# B&R Automation Studio project Lab3
Automation Studio 4.5.2.102

## Configuration SampleText

### Task classes (Cpu.sw)
```
Cyclic#1 (cycle 2000 us, tolerance 0 us):
  ncsdcctrl <- ncsdcctrl.prg
Cyclic#4:
  Program <- Program.prg
NcDataObjects: acp10etxen <- acp10etxen.dob, Axis_Xa <- Axis_Xobj.Axis_Xa.dob, Axis_Xi <- Axis_Xobj.Axis_Xi.dob
Libraries: Acp10sdc, sys_lib, Runtime, asstring, Acp10man, Acp10par, NcGlobal, Acp10_MC, brsystem, AsBrStr, Acp10sim, AsIOTime, Library
```

### Hardware
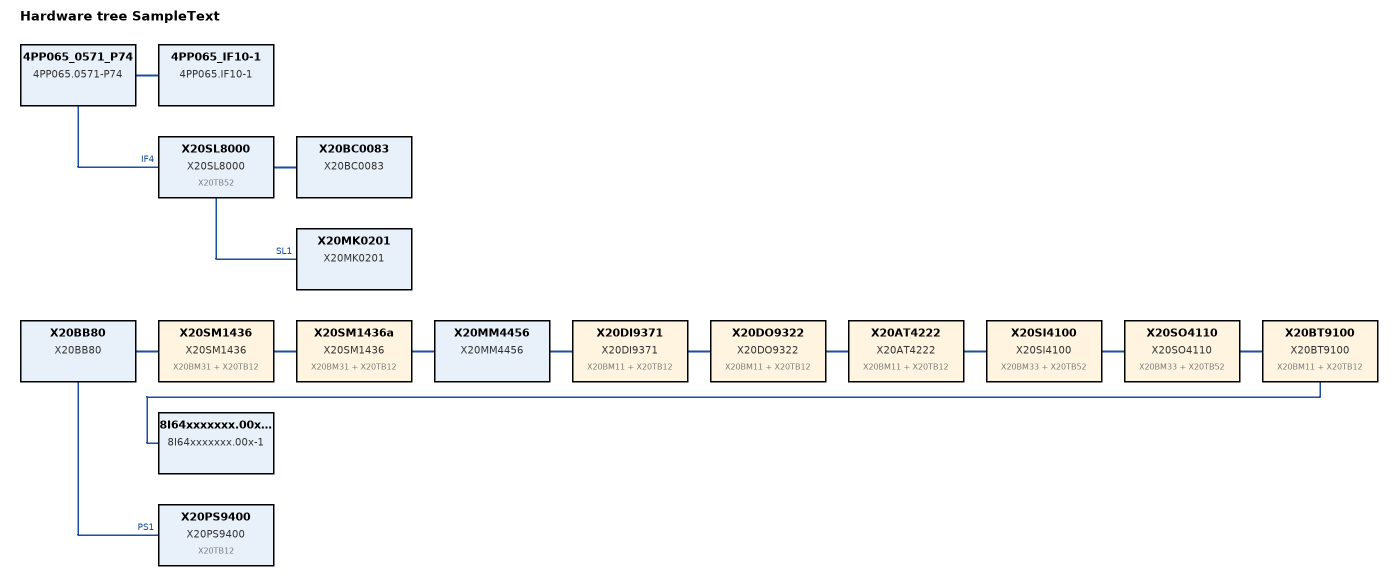
```
4PP065_0571_P74 : 4PP065.0571-P74 v1.1.2.0
  Connector IF4:
    EplInterfaceRedundant = 0
    EplEthInterfaceRedundant = 0
  Connector IF5:
    ActivateDevice = 1
    Mode = Manual
    InternetAddress = 10.1.1.13
    SubnetMask = 255.255.255.0
  ConfigurationID = DriveControl_SampleText
  Simulation = 1
  TimerDeviceType = EPLX2X
  TimerDevice = 4PP065_0571_P74.IF4
  TaskClassIdleTime = 2000
  Cyclic1Duration = 2000
  Cyclic1Tolerance = 0
  Cyclic1Output = 1
4PP065_IF10-1 : 4PP065.IF10-1 v1.0.3.0  [SS -> 4PP065_0571_P74.SS1]
8I64xxxxxxx.00x-1 : 8I64xxxxxxx.00x-1 v1.3.9.1  [X2X1 -> X20BT9100.X2X1 [Cable Type=X2XCable, Length=10, Version=1.0.0.2]]
X20AT4222 : X20AT4222 v1.2.3.0  [SS1 -> X20TB12e.SS; SL -> X20BM11c.SL1]
X20BB80 : X20BB80 v1.0.2.0
X20BC0083 : X20BC0083 v2.7.0.0  [PLK1 -> X20SL8000.PLK2 [Cable Type=PowerlinkCable, Length=10, Version=1.0.0.2]; SL -> X20BB80.SL1]
X20BM11 : X20BM11 v1.0.0.1  [X2X1 -> X20BM33a.X2X2]
X20BM11a : X20BM11 v1.0.0.1  [X2X1 -> X20MM4456.X2X2]
X20BM11b : X20BM11 v1.0.0.1  [X2X1 -> X20BM11a.X2X2]
X20BM11c : X20BM11 v1.0.0.1  [X2X1 -> X20BM11b.X2X2]
X20BM31 : X20BM31 v1.0.0.1  [X2X1 -> X20BB80.IF1]
X20BM31a : X20BM31 v1.0.0.1  [X2X1 -> X20BM31.X2X2]
X20BM33 : X20BM33 v1.0.0.4  [X2X1 -> X20BM11c.X2X2]
X20BM33a : X20BM33 v1.0.0.4  [X2X1 -> X20BM33.X2X2]
X20BT9100 : X20BT9100 v1.0.3.0  [SS1 -> X20TB12f.SS; SL -> X20BM11.SL1]
X20DI9371 : X20DI9371 v1.0.2.0  [SS1 -> X20TB12c.SS; SL -> X20BM11a.SL1]
X20DO9322 : X20DO9322 v1.0.3.0  [SS1 -> X20TB12d.SS; SL -> X20BM11b.SL1]
X20MK0201 : X20MK0201 v1.0.0.0  [SL -> X20SL8000.SL1]
X20MM4456 : X20MM4456 v1.1.5.0  [X2X1 -> X20BM31a.X2X2]
X20PS9400 : X20PS9400 v1.0.2.4  [SS1 -> X20TB12.SS; PS -> X20BB80.PS1]
X20SI4100 : X20SI4100 v1.10.1.1  [SS1 -> X20TB52.SS; SL -> X20BM33.SL1]
X20SL8000 : X20SL8000 v1.6.5.1  [PLK1 -> 4PP065_0571_P74.IF4 [Cable Type=PowerlinkCable, Length=10, Version=1.0.0.2]; PLK2 -> X20BC0083.PLK1 [Cable Type=PowerlinkCable, Length=10, Version=1.0.0.2]; SS1 -> X20TB52b.SS]
  SafeProject = SafeLOGIC-1
X20SM1436 : X20SM1436 v2.2.0.0  [SS1 -> X20TB12a.SS; SL -> X20BM31.SL1]
X20SM1436a : X20SM1436 v2.2.0.0  [SS1 -> X20TB12b.SS; SL -> X20BM31a.SL1]
X20SO4110 : X20SO4110 v1.10.1.1  [SS1 -> X20TB52a.SS; SL -> X20BM33a.SL1]
  SafeModuleID = 3
X20TB12 : X20TB12 v1.0.0.0
X20TB12a : X20TB12 v1.0.0.0
X20TB12b : X20TB12 v1.0.0.0
X20TB12c : X20TB12 v1.0.0.0
X20TB12d : X20TB12 v1.0.0.0
X20TB12e : X20TB12 v1.0.0.0
X20TB12f : X20TB12 v1.0.0.0
X20TB52 : X20TB52 v1.0.0.1
X20TB52a : X20TB52 v1.0.0.1
X20TB52b : X20TB52 v1.0.0.1
```

### IoMap.iom - 4PP065_0571_P74/IoMap.iom
```iecst
VAR_CONFIG
	Cyclic#1.Axis_X_DrvIf.iLifeCnt AT %IB."8I64xxxxxxx.00x-1".SDC_LifeCnt;
	Cyclic#1.Axis_X_DrvIf.iDrvOK AT %IX."8I64xxxxxxx.00x-1".ETAD_Input_Bool_02;
	Cyclic#1.Axis_X_DrvIf.oSetTime AT %QW."8I64xxxxxxx.00x-1".SDC_SetTime;
	Cyclic#1.Axis_X_DrvIf.oSetPos AT %QW."8I64xxxxxxx.00x-1".LFRD_Output;
	Cyclic#1.Axis_X_DiDoIf.iLifeCntDriveReady AT %IB."8I64xxxxxxx.00x-1".SDC_LifeCnt;
	Cyclic#1.Axis_X_DiDoIf.iLifeCntDriveEnable AT %IB."8I64xxxxxxx.00x-1".SDC_LifeCnt;
	Cyclic#1.Axis_X_DiDoIf.oDriveEnable AT %QX."8I64xxxxxxx.00x-1".CMDD_Output_Bool_00;
	Cyclic#1.Axis_X_ModuleOk AT %QX."8I64xxxxxxx.00x-1".CMDD_Output_Bool_01;
	Cyclic#1.Axis_X_ModuleOk AT %QX."8I64xxxxxxx.00x-1".CMDD_Output_Bool_02;
	Cyclic#1.Axis_X_ModuleOk AT %IX."8I64xxxxxxx.00x-1".ModuleOk;
	Cyclic#1.Axis_X_DiDoIf.oDriveEnable AT %QX."8I64xxxxxxx.00x-1".CMDD_Output_Bool_03;
	Cyclic#1.Axis_X_DiDoIf.iDriveReady AT %IX."8I64xxxxxxx.00x-1".ETAD_Input_Bool_02;
	::Program:coil_powered AT %IX."X20DI9371".DigitalInput01;
	::Program:axis_X.pwm_value AT %QW."X20MM4456".PulseWidthCurrentPWM01;
	::Program:axis_X.reset_error  AT %QX."X20MM4456".ClearError01;
	::Program:axis_X.endswitch_a_reached  AT %IX."X20MM4456".StatusInput03;
	::Program:axis_X.endswitch_b_reached AT %IX."X20MM4456".StatusInput04;
	::Program:axis_X.counter AT %IW."X20MM4456".Counter01;
	::Program:pwm_period  AT %QW."X20MM4456".PeriodDurationPWM;
	::Program:axis_X.reset_counter AT %QX."X20MM4456".ResetCounter01;
	::Program:coil_pwm_value  AT %QW."X20MM4456".PulseWidthCurrentPWM04;
END_VAR
```

### Acp10map.ncm - 4PP065_0571_P74/Motion/Acp10map.ncm
```
NcMapping (NcSwId=Acp10, DisabledNodesAreHidden=False)
  NcObject Axis_X (ModuleId=8I64xxxxxxx.00x-1, ModuleAddress=SDC_IF1.ST2, Type=ncAXIS, Channel=1, AcoposSimulation=Off, InitParameter=Axis_Xi, AcoposParameter=Axis_Xa, Disabled=FALSE, ModuleDisabled=FALSE)
```

## Logical view

### Axis_Xi.ax
```
InitParameter (Version=5.02.1, NcSwId=Acp10)
  ACP10AXIS_typ:
    dig_in:
      level:
        reference = ncACTIV_HI
        pos_hw_end = ncACTIV_HI
        neg_hw_end = ncACTIV_HI
        trigger1 = ncACTIV_HI
        trigger2 = ncACTIV_LO + ncQUICKSTOP
    encoder_if:
      parameter:
        count_dir = ncSTANDARD
        scaling:
          load:
            units = 3000
            rev_motor = 1
    limit:
      parameter:
        v_pos = 10000
        v_neg = 10000
        a1_pos = 10000.0
        a2_pos = 10000.0
        a1_neg = 10000.0
        a2_neg = 10000.0
        t_jolt = 0
        t_in_pos = 0
        pos_sw_end = 2000000000
        neg_sw_end = -2000000000
        ds_warning = 500
        ds_stop = 50000.0
        a_stop = 1.0e30
        dv_stop = 0
        dv_stop_mode = ncOFF
    controller:
      mode = ncPOSITION
      position:
        kv = 10.0
        tn = 0
        t_predict = 0.01
        t_total = 0.01
        p_max = 1.0e30
        i_max = 0
      speed:
        kv = 2.0
        tn = 0
        t_filter = 0.0
        isq_filter1:
          type = ncOFF
          a0 = 0.0
          a1 = 0.0
          b0 = 0.0
          b1 = 0.0
          b2 = 0.0
          c0_par_id = 0
          c1_par_id = 0
        isq_filter2:
          type = ncOFF
          a0 = 0.0
          a1 = 0.0
          b0 = 0.0
          b1 = 0.0
          b2 = 0.0
          c0_par_id = 0
          c1_par_id = 0
        isq_filter3:
          type = ncOFF
          a0 = 0.0
          a1 = 0.0
          b0 = 0.0
          b1 = 0.0
          b2 = 0.0
          c0_par_id = 0
          c1_par_id = 0
      uf:
        type = ncLINEAR + ncCORRECTION
        auto_config = ncMOTOR_PAR
        u0 = 0
        un = 0
        fn = 50.0
        k_f_slip = 0
      ff:
        torque_load = 0.0
        torque_pos = 0.0
        torque_neg = 0.0
        kv_torque = 0.0
        inertia = 0.0
        t_filter_a = 0.0
    move:
      stop:
        parameter[0]:
          decel_ramp = ncA_LIMIT
          controller = ncON
        parameter[1]:
          decel_ramp = ncA_LIMIT
          controller = ncON
        parameter[2]:
          decel_ramp = ncA_LIMIT
          controller = ncON
        parameter[3]:
          decel_ramp = ncA_LIMIT
          controller = ncON
        quickstop:
          decel_ramp = ncA_LIMIT
          t_jolt = 0
        drive_error:
          decel_ramp = ncA_LIMIT
      homing:
        parameter:
          s = 0
          v_switch = 6000.0
          v_trigger = 2000.0
          a = 10000.0
          mode = ncEND_SWITCH
          edge_sw = ncNEGATIVE
          start_dir = ncPOSITIVE
          trigg_dir = ncPOSITIVE
          ref_pulse = ncOFF
          fix_dir = ncOFF
          tr_s_block = 0
          torque_lim = 0
          ds_block = 0
          ds_stop = 0
      basis:
        parameter:
          v_pos = 5000
          v_neg = 5000
          a1_pos = 50000
          a2_pos = 50000
          a1_neg = 50000
          a2_neg = 50000
    message:
      text:
        parameter:
          format = ncBREAK
          columns = 80
          data_modul = acp10etxen
```

### Program Logical/ncsdcctrl

#### ncsdcctrlCyclic.st
```iecst
PROGRAM _CYCLIC

(* ### BEGIN Axis_X ### *)

(* life counter emulation of digital inputs *)
        Axis_X_DiDoIf.iLifeCntReference := Axis_X_DiDoIf.iLifeCntReference + 1;
        Axis_X_DiDoIf.iLifeCntNegHwEnd  := Axis_X_DiDoIf.iLifeCntNegHwEnd  + 1;
        Axis_X_DiDoIf.iLifeCntPosHwEnd  := Axis_X_DiDoIf.iLifeCntPosHwEnd  + 1;

(* ### END Axis_X ### *)

END_PROGRAM
```

#### ncsdcctrlInit.st
```iecst
PROGRAM _INIT

(* ### BEGIN Axis_X ### *)

(* initialize variables *)
        Axis_X_HW.DrvIf_Typ := ncSDC_DRVSERVO16;
        brsstrcpy(ADR(Axis_X_HW.DrvIf_Name[0]), ADR('Axis_X_DrvIf'));
        Axis_X_HW.DiDoIf_Typ := ncSDC_DIDO;
        brsstrcpy(ADR(Axis_X_HW.DiDoIf_Name[0]), ADR('Axis_X_DiDoIf'));

(* force variable offset generation *)
        Axis_X.size                      := Axis_X.size;
        Axis_X_DrvIf.iLifeCnt            := Axis_X_DrvIf.iLifeCnt;
        Axis_X_DiDoIf.iLifeCntDriveReady := Axis_X_DiDoIf.iLifeCntDriveReady;
        Axis_X_ModuleOk                  := Axis_X_ModuleOk;

(* assign your hardware inputs here*)

(*      Axis_X_DiDoIf.iPosHwEnd  := Axis_X_DiDoIf.iPosHwEnd;
        Axis_X_DiDoIf.iNegHwEnd  := Axis_X_DiDoIf.iNegHwEnd;
        Axis_X_DiDoIf.iReference := Axis_X_DiDoIf.iReference;
 *)

(* ### END Axis_X ### *)

END_PROGRAM
```

### Program Logical/Program

#### Variables.var
```iecst
VAR
	coil_pwm_value : INT := 0;
	coil_powered : BOOL := FALSE;
	axis_X : FB_Axis := (0);
	pwm_period : UINT := 0;
	fb_controller : FB_controller := (0);
	XNegHwEnd : REAL := 0.0;
	XPosHwEnd : REAL := 0.0;
	enable : BOOL := FALSE;
	fb_motor : FB_Motor := (0);
END_VAR
```

#### Main.cpp
```cpp
#include <bur/plctypes.h>

#ifdef _DEFAULT_INCLUDES
	#include <AsDefault.h>
#endif

// amount of memory to be allocated for heap storage must be specified for every ANSI C++ program with the bur_heap_size variable
unsigned long bur_heap_size = 0xFFFF;

void _INIT ProgramInit(void)
{
	// Insert code here
	Axis_X_HW.EncIf1_Typ = ncSDC_ENC16;
	Axis_X_HW.DiDoIf_Typ = ncSDC_DIDO;
	Axis_X_HW.DrvIf_Typ = ncSDC_DRVSERVO16;
	//strcpy(Axis_X_HW.EncIf1_Name, "Axis_X_EncIf");
	//strcpy(Axis_X_HW.DrvIf_Name, "Axis_X_DrvIf");
	//strcpy(Axis_X_HW.DiDoIf_Name, "Axis_X_DiDoIf");

	Axis_X_ModuleOk = 1;
	Axis_X_EncIf.iEncOK = 1;
	Axis_X_DrvIf.iDrvOK = 1;
	Axis_X_DrvIf.iStatusEnable = 1;
	Axis_X_DiDoIf.iDriveReady = 1;

	axis_X.last_counter = 0;
	axis_X.counter = axis_X.last_counter;
	pwm_period = 0.05;
	axis_X.pwm_period = pwm_period;

	axis_X.fb_controller.dt = 0.002;
	axis_X.fb_controller.integrator.dt = 0.002;
	axis_X.fb_controller.k_i = 0.0072;
	axis_X.fb_controller.k_p = 0.0072;
	axis_X.fb_controller.max_abs_value = 40.0;

	fb_motor.dt = 0.01;
	fb_motor.ke = 1;
	fb_motor.Tm = 0.1;
	fb_motor.u = 0;
	fb_motor.phi = 0;
	fb_motor.integrator.dt = 0.01;

}

void _CYCLIC ProgramCyclic(void)
{
	// Insert code here
	Axis_X_EncIf.iLifeCnt++;
	Axis_X_EncIf.iActTime = (INT)AsIOTimeCyclicStart();
	Axis_X_DrvIf.iLifeCnt++;
	Axis_X_DrvIf.oSetPos = Axis_X.monitor.v;
	Axis_X_DiDoIf.iLifeCntDriveEnable++;
	Axis_X_DiDoIf.iLifeCntDriveReady++;
	Axis_X_DiDoIf.iLifeCntNegHwEnd++;
	Axis_X_DiDoIf.iLifeCntPosHwEnd++;
	Axis_X_DiDoIf.iLifeCntReference++;

	axis_X.iActPos = Axis_X_EncIf.iActPos;
	axis_X.iLifeCnt = Axis_X_EncIf.iLifeCnt;
	axis_X.iNegHwEnd = Axis_X_DiDoIf.iNegHwEnd;
	axis_X.iPosHwEnd = Axis_X_DiDoIf.iPosHwEnd;
	axis_X.oSetPos = Axis_X_DrvIf.oSetPos;

	FB_Axis(&axis_X);

	Axis_X_EncIf.iActPos = axis_X.iActPos;
	Axis_X_EncIf.iLifeCnt = axis_X.iLifeCnt;
	Axis_X_DiDoIf.iNegHwEnd = axis_X.iNegHwEnd;
	Axis_X_DiDoIf.iPosHwEnd = axis_X.iPosHwEnd;
	Axis_X_DrvIf.oSetPos = axis_X.oSetPos;

	if(Axis_X_DrvIf.oSetPos != 0)
	{
		fb_motor.u = axis_X.pwm_value / axis_X.pwm_period * 32767;
		FB_Motor(&fb_motor);
		axis_X.counter = fb_motor.phi;

		axis_X.endswitch_a_reached = axis_X.counter <= -3000 ? 1 : 0;
		axis_X.endswitch_b_reached = axis_X.counter >= 3000 ? 1 : 0;
	}

}

void _EXIT ProgramExit(void)
{
	// Insert code here

}
```
